(* Schneider Machine Expert - Basic project tank_level_1m_TM221CE24T, file version 3.0.0.0 *)
(* ProjectInformations: Name=Tank Level Control 1m - Ultrasonic, Version=1.0, LastModified=2025-12-26, Author=PLCAutoPilot, Description=Automatic tank level control with ultrasonic sensor (4-20mA), TM3AI4 expansion, inlet/outlet valves with hysteresis *)

HARDWARE
  Cpu 0: TM221CE24T
  ModuleExtensionObject 0: TM3AI4/G
  EthernetConfiguration: NetworkName=M221, IpAllocationMode=FixedAddress, IpAddress=0.0.0.0, SubnetMask=0.0.0.0
  SerialLineConfiguration: Baud=Baud19200, Parity=ParityEven, DataBits=DataBits8, StopBits=StopBits1, PhysicalMedium=PhysicalMediumRs485, TransmissionMode=TransmissionModeModbusRtu, SlaveId=1, Addressing=SlaveAddressing
  MastTask: UsePeriodScanMode=false, PeriodScan=100
  FastTask: Period=255
  CpuBehavior: StartingMode=StartAsPreviousState, AutoSaveRamOnEeprom=true, WatchdogPeriod=250

SYMBOLS  (address, symbol, comment, settings)
  %S12      SB_RUNMODE  "The controller is running"
  %IW1.0    TANK_LEVEL  [Type=Type_4_20mA, Scope=Scope_Customized, Minimum=300, Maximum=3000]

POU Tank Level Control 1m
  (* SectionNumber=0 *)

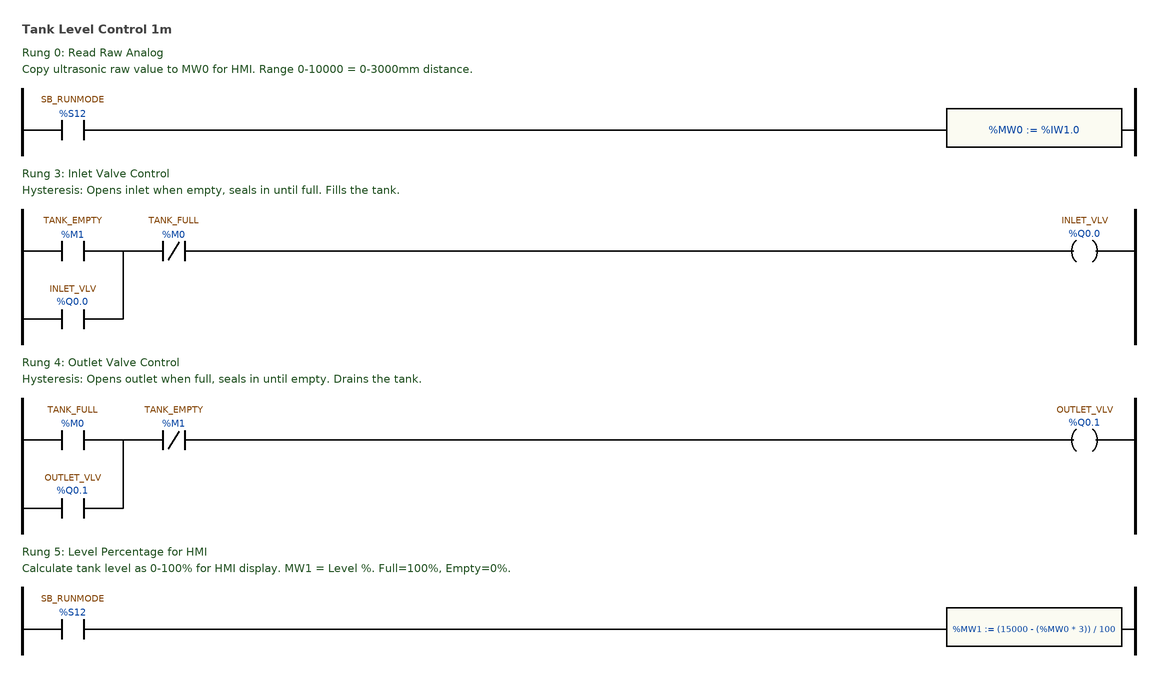

// Rung 0: Read Raw Analog
// Copy ultrasonic raw value to MW0 for HMI. Range 0-10000 = 0-3000mm distance.
  LD %S12                 (* SB_RUNMODE *)
  [ %MW0 := %IW1.0 ]      (* TANK_LEVEL *)
  // as ST:
  //   IF SB_RUNMODE THEN %MW0 := TANK_LEVEL; END_IF;

// Rung 1: Tank Full Detection
// Tank FULL when distance less than 540mm (raw 1800). Level above 960mm.
  LD [%IW1.0<1800]        (* TANK_LEVEL *)
  ST %M0
  // as ST:
  //   %M0 := TANK_LEVEL<1800;
  (* the ladder stored for this rung does not match its IL; not drawn *)

// Rung 2: Tank Empty Detection
// Tank EMPTY when distance more than 1440mm (raw 4800). Level below 60mm.
  LD [%IW1.0>4800]        (* TANK_LEVEL *)
  ST %M1
  // as ST:
  //   %M1 := TANK_LEVEL>4800;
  (* the ladder stored for this rung does not match its IL; not drawn *)

// Rung 3: Inlet Valve Control
// Hysteresis: Opens inlet when empty, seals in until full. Fills the tank.
  LD %M1
  OR %Q0.0
  ANDN %M0
  ST %Q0.0
  // as ST:
  //   %Q0.0 := (%M1 OR %Q0.0) AND NOT %M0;

// Rung 4: Outlet Valve Control
// Hysteresis: Opens outlet when full, seals in until empty. Drains the tank.
  LD %M0
  OR %Q0.1
  ANDN %M1
  ST %Q0.1
  // as ST:
  //   %Q0.1 := (%M0 OR %Q0.1) AND NOT %M1;

// Rung 5: Level Percentage for HMI
// Calculate tank level as 0-100% for HMI display. MW1 = Level %. Full=100%, Empty=0%.
  LD %S12                 (* SB_RUNMODE *)
  [ %MW1 := (15000 - (%MW0 * 3)) / 100 ]
  // as ST:
  //   IF SB_RUNMODE THEN %MW1 := (15000 - (%MW0 * 3)) / 100; END_IF;
